{attribute addProperty BoxType "EL6080-0000-0016"}
{attribute addProperty Id "StatusAT %I*ARRAY [0..1] OF USINT00"}
{attribute addProperty CRC "2008604244"}
{attribute addProperty SizeInBites "0"}
{attribute addProperty SizeInBytes "0"}
TYPE Status_77B8DE54 :
STRUCT
	{attribute addProperty Name "Status"}
	Status AT %I* : ARRAY [0..1] OF USINT;
END_STRUCT
END_TYPE

(* stored: Version 1.2.0.0, ProductVersion 3.1.4024.9
   DUT Status_77B8DE54: Id {b99db28d-ef0f-45af-b074-4b30ad2102e0} *)
